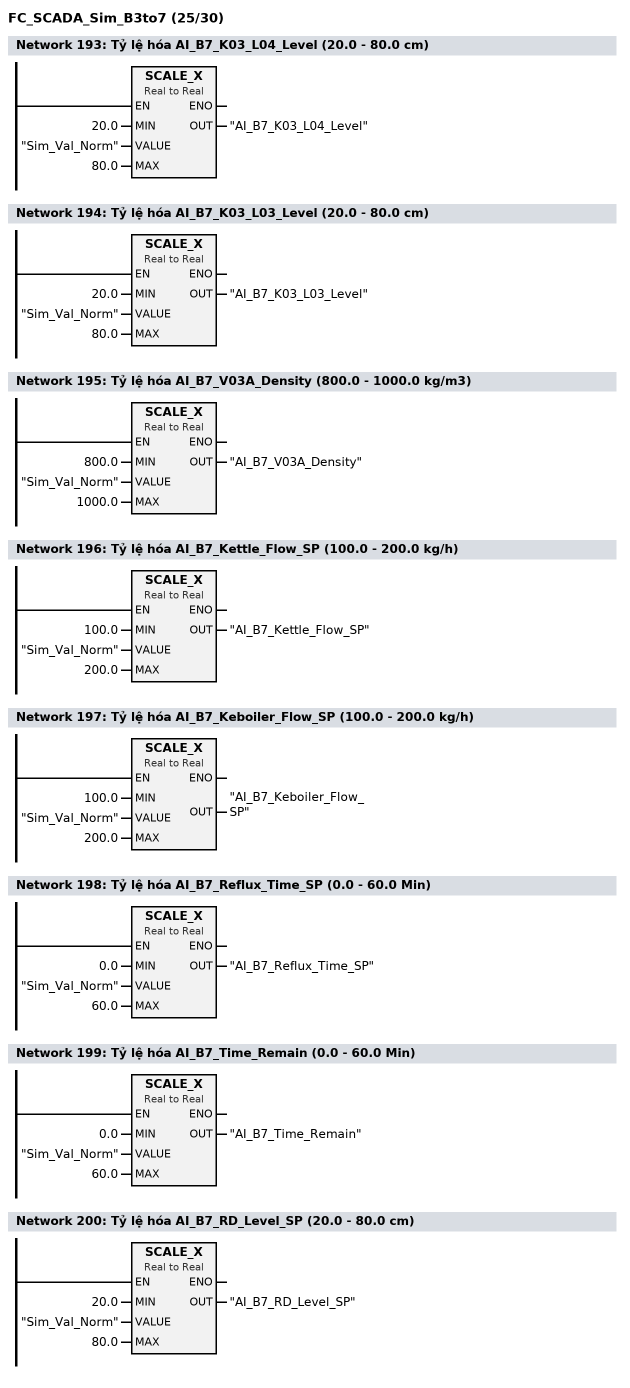
   RUNG wire#powerrail
      { S7_Templates := "[SrcType := Real, DestType := Real]" } Scale(min := 20.0, value := "Sim_Val_Norm", max := 80.0, out => "AI_B7_K03_L04_Level")
   END_RUNG
   // the same network as SCL:
   "AI_B7_K03_L04_Level" := SCALE_X(MIN := 20.0, VALUE := "Sim_Val_Norm", MAX := 80.0);
END_REGION

REGION Network 194: Tỷ lệ hóa AI_B7_K03_L03_Level (20.0 - 80.0 cm)
   RUNG wire#powerrail
      { S7_Templates := "[SrcType := Real, DestType := Real]" } Scale(min := 20.0, value := "Sim_Val_Norm", max := 80.0, out => "AI_B7_K03_L03_Level")
   END_RUNG
   // the same network as SCL:
   "AI_B7_K03_L03_Level" := SCALE_X(MIN := 20.0, VALUE := "Sim_Val_Norm", MAX := 80.0);
END_REGION

REGION Network 195: Tỷ lệ hóa AI_B7_V03A_Density (800.0 - 1000.0 kg/m3)
   RUNG wire#powerrail
      { S7_Templates := "[SrcType := Real, DestType := Real]" } Scale(min := 800.0, value := "Sim_Val_Norm", max := 1000.0, out => "AI_B7_V03A_Density")
   END_RUNG
   // the same network as SCL:
   "AI_B7_V03A_Density" := SCALE_X(MIN := 800.0, VALUE := "Sim_Val_Norm", MAX := 1000.0);
END_REGION

REGION Network 196: Tỷ lệ hóa AI_B7_Kettle_Flow_SP (100.0 - 200.0 kg/h)
   RUNG wire#powerrail
      { S7_Templates := "[SrcType := Real, DestType := Real]" } Scale(min := 100.0, value := "Sim_Val_Norm", max := 200.0, out => "AI_B7_Kettle_Flow_SP")
   END_RUNG
   // the same network as SCL:
   "AI_B7_Kettle_Flow_SP" := SCALE_X(MIN := 100.0, VALUE := "Sim_Val_Norm", MAX := 200.0);
END_REGION

REGION Network 197: Tỷ lệ hóa AI_B7_Keboiler_Flow_SP (100.0 - 200.0 kg/h)
   RUNG wire#powerrail
      { S7_Templates := "[SrcType := Real, DestType := Real]" } Scale(min := 100.0, value := "Sim_Val_Norm", max := 200.0, out => "AI_B7_Keboiler_Flow_SP")
   END_RUNG
   // the same network as SCL:
   "AI_B7_Keboiler_Flow_SP" := SCALE_X(MIN := 100.0, VALUE := "Sim_Val_Norm", MAX := 200.0);
END_REGION

REGION Network 198: Tỷ lệ hóa AI_B7_Reflux_Time_SP (0.0 - 60.0 Min)
   RUNG wire#powerrail
      { S7_Templates := "[SrcType := Real, DestType := Real]" } Scale(min := 0.0, value := "Sim_Val_Norm", max := 60.0, out => "AI_B7_Reflux_Time_SP")
   END_RUNG
   // the same network as SCL:
   "AI_B7_Reflux_Time_SP" := SCALE_X(MIN := 0.0, VALUE := "Sim_Val_Norm", MAX := 60.0);
END_REGION

REGION Network 199: Tỷ lệ hóa AI_B7_Time_Remain (0.0 - 60.0 Min)
   RUNG wire#powerrail
      { S7_Templates := "[SrcType := Real, DestType := Real]" } Scale(min := 0.0, value := "Sim_Val_Norm", max := 60.0, out => "AI_B7_Time_Remain")
   END_RUNG
   // the same network as SCL:
   "AI_B7_Time_Remain" := SCALE_X(MIN := 0.0, VALUE := "Sim_Val_Norm", MAX := 60.0);
END_REGION

REGION Network 200: Tỷ lệ hóa AI_B7_RD_Level_SP (20.0 - 80.0 cm)
   RUNG wire#powerrail
      { S7_Templates := "[SrcType := Real, DestType := Real]" } Scale(min := 20.0, value := "Sim_Val_Norm", max := 80.0, out => "AI_B7_RD_Level_SP")
   END_RUNG
   // the same network as SCL:
   "AI_B7_RD_Level_SP" := SCALE_X(MIN := 20.0, VALUE := "Sim_Val_Norm", MAX := 80.0);
END_REGION

REGION Network 201: Tỷ lệ hóa AI_B7_Reflux_Flow_SP (100.0 - 200.0 L/h)
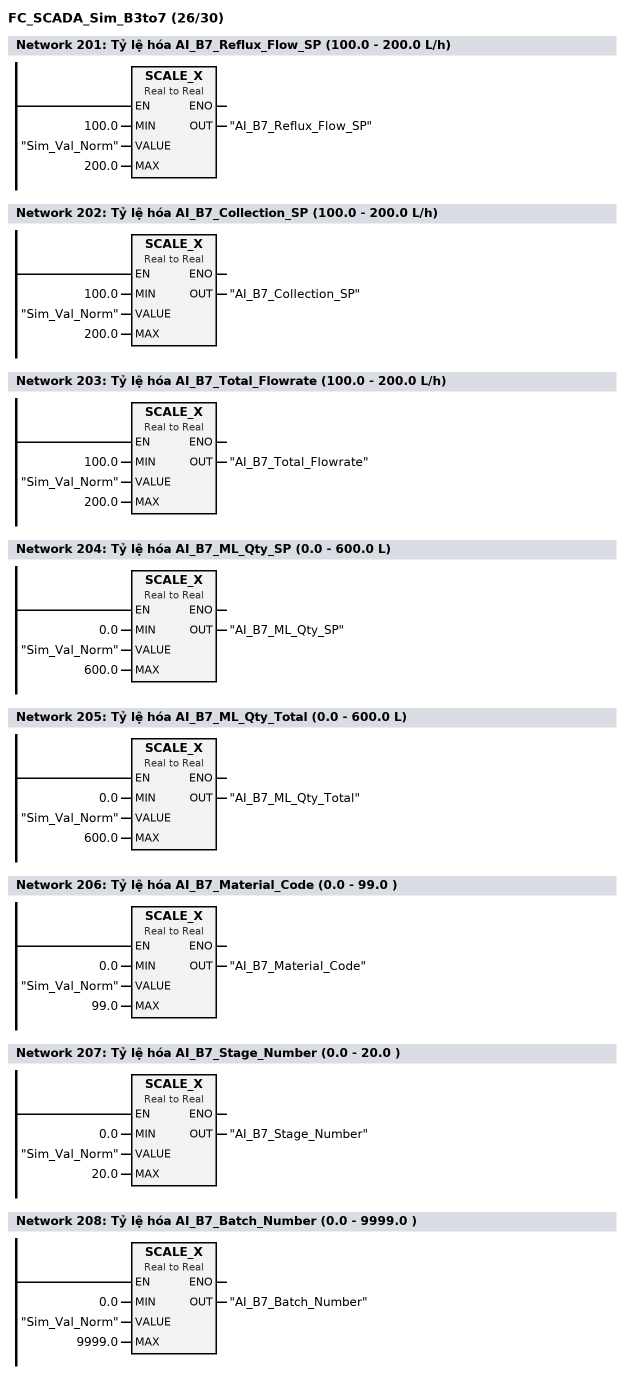
   RUNG wire#powerrail
      { S7_Templates := "[SrcType := Real, DestType := Real]" } Scale(min := 100.0, value := "Sim_Val_Norm", max := 200.0, out => "AI_B7_Reflux_Flow_SP")
   END_RUNG
   // the same network as SCL:
   "AI_B7_Reflux_Flow_SP" := SCALE_X(MIN := 100.0, VALUE := "Sim_Val_Norm", MAX := 200.0);
END_REGION

REGION Network 202: Tỷ lệ hóa AI_B7_Collection_SP (100.0 - 200.0 L/h)
   RUNG wire#powerrail
      { S7_Templates := "[SrcType := Real, DestType := Real]" } Scale(min := 100.0, value := "Sim_Val_Norm", max := 200.0, out => "AI_B7_Collection_SP")
   END_RUNG
   // the same network as SCL:
   "AI_B7_Collection_SP" := SCALE_X(MIN := 100.0, VALUE := "Sim_Val_Norm", MAX := 200.0);
END_REGION

REGION Network 203: Tỷ lệ hóa AI_B7_Total_Flowrate (100.0 - 200.0 L/h)
   RUNG wire#powerrail
      { S7_Templates := "[SrcType := Real, DestType := Real]" } Scale(min := 100.0, value := "Sim_Val_Norm", max := 200.0, out => "AI_B7_Total_Flowrate")
   END_RUNG
   // the same network as SCL:
   "AI_B7_Total_Flowrate" := SCALE_X(MIN := 100.0, VALUE := "Sim_Val_Norm", MAX := 200.0);
END_REGION

REGION Network 204: Tỷ lệ hóa AI_B7_ML_Qty_SP (0.0 - 600.0 L)
   RUNG wire#powerrail
      { S7_Templates := "[SrcType := Real, DestType := Real]" } Scale(min := 0.0, value := "Sim_Val_Norm", max := 600.0, out => "AI_B7_ML_Qty_SP")
   END_RUNG
   // the same network as SCL:
   "AI_B7_ML_Qty_SP" := SCALE_X(MIN := 0.0, VALUE := "Sim_Val_Norm", MAX := 600.0);
END_REGION

REGION Network 205: Tỷ lệ hóa AI_B7_ML_Qty_Total (0.0 - 600.0 L)
   RUNG wire#powerrail
      { S7_Templates := "[SrcType := Real, DestType := Real]" } Scale(min := 0.0, value := "Sim_Val_Norm", max := 600.0, out => "AI_B7_ML_Qty_Total")
   END_RUNG
   // the same network as SCL:
   "AI_B7_ML_Qty_Total" := SCALE_X(MIN := 0.0, VALUE := "Sim_Val_Norm", MAX := 600.0);
END_REGION

REGION Network 206: Tỷ lệ hóa AI_B7_Material_Code (0.0 - 99.0 )
   RUNG wire#powerrail
      { S7_Templates := "[SrcType := Real, DestType := Real]" } Scale(min := 0.0, value := "Sim_Val_Norm", max := 99.0, out => "AI_B7_Material_Code")
   END_RUNG
   // the same network as SCL:
   "AI_B7_Material_Code" := SCALE_X(MIN := 0.0, VALUE := "Sim_Val_Norm", MAX := 99.0);
END_REGION

REGION Network 207: Tỷ lệ hóa AI_B7_Stage_Number (0.0 - 20.0 )
   RUNG wire#powerrail
      { S7_Templates := "[SrcType := Real, DestType := Real]" } Scale(min := 0.0, value := "Sim_Val_Norm", max := 20.0, out => "AI_B7_Stage_Number")
   END_RUNG
   // the same network as SCL:
   "AI_B7_Stage_Number" := SCALE_X(MIN := 0.0, VALUE := "Sim_Val_Norm", MAX := 20.0);
END_REGION

REGION Network 208: Tỷ lệ hóa AI_B7_Batch_Number (0.0 - 9999.0 )
   RUNG wire#powerrail
      { S7_Templates := "[SrcType := Real, DestType := Real]" } Scale(min := 0.0, value := "Sim_Val_Norm", max := 9999.0, out => "AI_B7_Batch_Number")
   END_RUNG
   // the same network as SCL:
   "AI_B7_Batch_Number" := SCALE_X(MIN := 0.0, VALUE := "Sim_Val_Norm", MAX := 9999.0);
END_REGION

REGION Network 209: Tỷ lệ hóa AI_B7_Current_User_ID (0.0 - 999.0 )
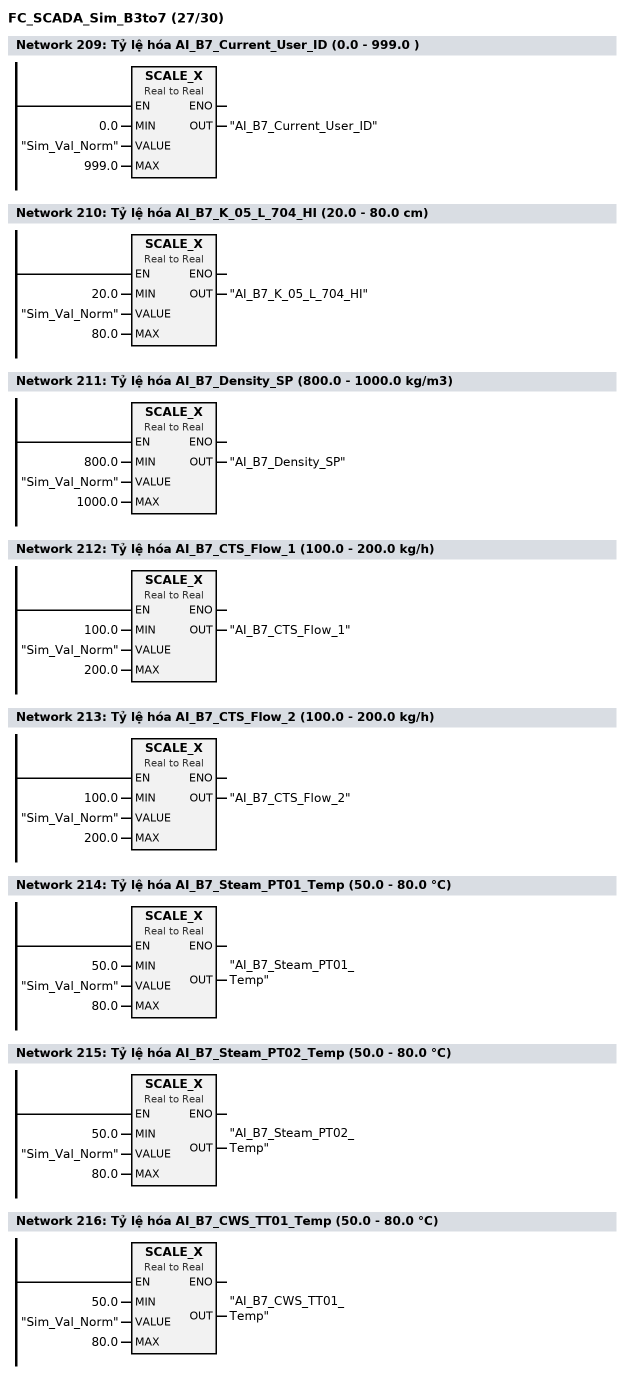
   RUNG wire#powerrail
      { S7_Templates := "[SrcType := Real, DestType := Real]" } Scale(min := 0.0, value := "Sim_Val_Norm", max := 999.0, out => "AI_B7_Current_User_ID")
   END_RUNG
   // the same network as SCL:
   "AI_B7_Current_User_ID" := SCALE_X(MIN := 0.0, VALUE := "Sim_Val_Norm", MAX := 999.0);
END_REGION

REGION Network 210: Tỷ lệ hóa AI_B7_K_05_L_704_HI (20.0 - 80.0 cm)
   RUNG wire#powerrail
      { S7_Templates := "[SrcType := Real, DestType := Real]" } Scale(min := 20.0, value := "Sim_Val_Norm", max := 80.0, out => "AI_B7_K_05_L_704_HI")
   END_RUNG
   // the same network as SCL:
   "AI_B7_K_05_L_704_HI" := SCALE_X(MIN := 20.0, VALUE := "Sim_Val_Norm", MAX := 80.0);
END_REGION

REGION Network 211: Tỷ lệ hóa AI_B7_Density_SP (800.0 - 1000.0 kg/m3)
   RUNG wire#powerrail
      { S7_Templates := "[SrcType := Real, DestType := Real]" } Scale(min := 800.0, value := "Sim_Val_Norm", max := 1000.0, out => "AI_B7_Density_SP")
   END_RUNG
   // the same network as SCL:
   "AI_B7_Density_SP" := SCALE_X(MIN := 800.0, VALUE := "Sim_Val_Norm", MAX := 1000.0);
END_REGION

REGION Network 212: Tỷ lệ hóa AI_B7_CTS_Flow_1 (100.0 - 200.0 kg/h)
   RUNG wire#powerrail
      { S7_Templates := "[SrcType := Real, DestType := Real]" } Scale(min := 100.0, value := "Sim_Val_Norm", max := 200.0, out => "AI_B7_CTS_Flow_1")
   END_RUNG
   // the same network as SCL:
   "AI_B7_CTS_Flow_1" := SCALE_X(MIN := 100.0, VALUE := "Sim_Val_Norm", MAX := 200.0);
END_REGION

REGION Network 213: Tỷ lệ hóa AI_B7_CTS_Flow_2 (100.0 - 200.0 kg/h)
   RUNG wire#powerrail
      { S7_Templates := "[SrcType := Real, DestType := Real]" } Scale(min := 100.0, value := "Sim_Val_Norm", max := 200.0, out => "AI_B7_CTS_Flow_2")
   END_RUNG
   // the same network as SCL:
   "AI_B7_CTS_Flow_2" := SCALE_X(MIN := 100.0, VALUE := "Sim_Val_Norm", MAX := 200.0);
END_REGION

REGION Network 214: Tỷ lệ hóa AI_B7_Steam_PT01_Temp (50.0 - 80.0 °C)
   RUNG wire#powerrail
      { S7_Templates := "[SrcType := Real, DestType := Real]" } Scale(min := 50.0, value := "Sim_Val_Norm", max := 80.0, out => "AI_B7_Steam_PT01_Temp")
   END_RUNG
   // the same network as SCL:
   "AI_B7_Steam_PT01_Temp" := SCALE_X(MIN := 50.0, VALUE := "Sim_Val_Norm", MAX := 80.0);
END_REGION

REGION Network 215: Tỷ lệ hóa AI_B7_Steam_PT02_Temp (50.0 - 80.0 °C)
   RUNG wire#powerrail
      { S7_Templates := "[SrcType := Real, DestType := Real]" } Scale(min := 50.0, value := "Sim_Val_Norm", max := 80.0, out => "AI_B7_Steam_PT02_Temp")
   END_RUNG
   // the same network as SCL:
   "AI_B7_Steam_PT02_Temp" := SCALE_X(MIN := 50.0, VALUE := "Sim_Val_Norm", MAX := 80.0);
END_REGION

REGION Network 216: Tỷ lệ hóa AI_B7_CWS_TT01_Temp (50.0 - 80.0 °C)
   RUNG wire#powerrail
      { S7_Templates := "[SrcType := Real, DestType := Real]" } Scale(min := 50.0, value := "Sim_Val_Norm", max := 80.0, out => "AI_B7_CWS_TT01_Temp")
   END_RUNG
   // the same network as SCL:
   "AI_B7_CWS_TT01_Temp" := SCALE_X(MIN := 50.0, VALUE := "Sim_Val_Norm", MAX := 80.0);
END_REGION

REGION Network 217: Tỷ lệ hóa AI_B7_CWS_TT02_Temp (50.0 - 80.0 °C)
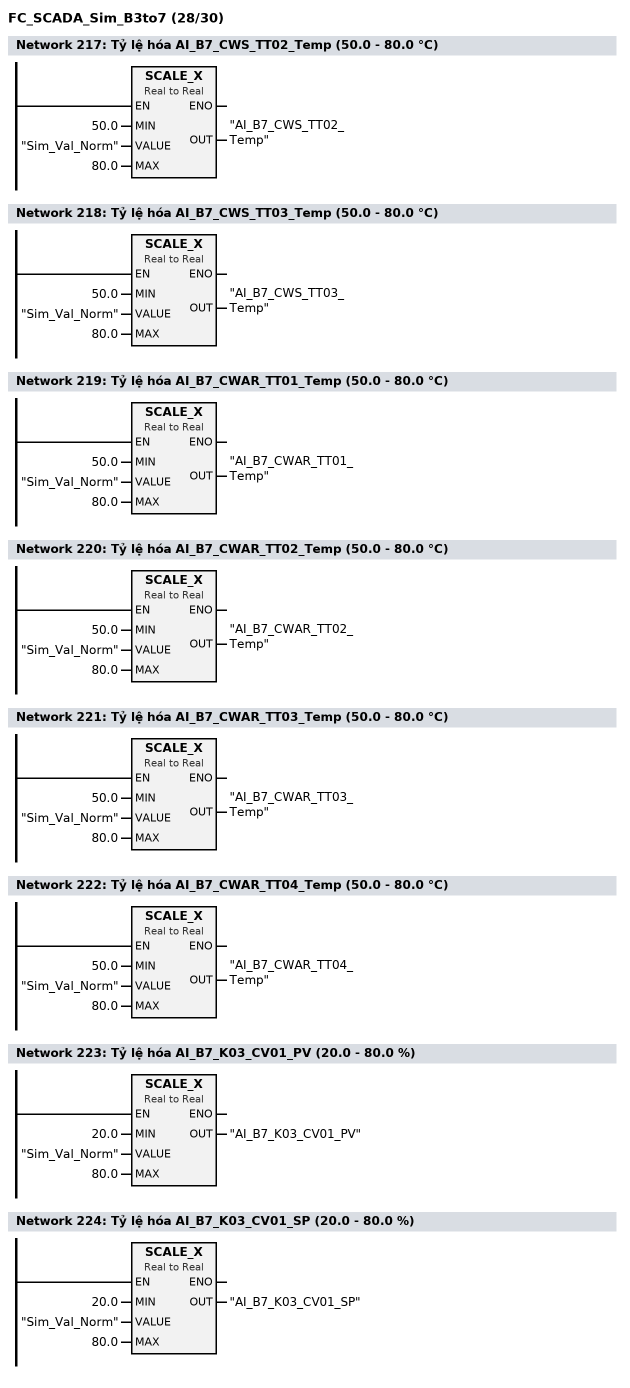
   RUNG wire#powerrail
      { S7_Templates := "[SrcType := Real, DestType := Real]" } Scale(min := 50.0, value := "Sim_Val_Norm", max := 80.0, out => "AI_B7_CWS_TT02_Temp")
   END_RUNG
   // the same network as SCL:
   "AI_B7_CWS_TT02_Temp" := SCALE_X(MIN := 50.0, VALUE := "Sim_Val_Norm", MAX := 80.0);
END_REGION

REGION Network 218: Tỷ lệ hóa AI_B7_CWS_TT03_Temp (50.0 - 80.0 °C)
   RUNG wire#powerrail
      { S7_Templates := "[SrcType := Real, DestType := Real]" } Scale(min := 50.0, value := "Sim_Val_Norm", max := 80.0, out => "AI_B7_CWS_TT03_Temp")
   END_RUNG
   // the same network as SCL:
   "AI_B7_CWS_TT03_Temp" := SCALE_X(MIN := 50.0, VALUE := "Sim_Val_Norm", MAX := 80.0);
END_REGION

REGION Network 219: Tỷ lệ hóa AI_B7_CWAR_TT01_Temp (50.0 - 80.0 °C)
   RUNG wire#powerrail
      { S7_Templates := "[SrcType := Real, DestType := Real]" } Scale(min := 50.0, value := "Sim_Val_Norm", max := 80.0, out => "AI_B7_CWAR_TT01_Temp")
   END_RUNG
   // the same network as SCL:
   "AI_B7_CWAR_TT01_Temp" := SCALE_X(MIN := 50.0, VALUE := "Sim_Val_Norm", MAX := 80.0);
END_REGION

REGION Network 220: Tỷ lệ hóa AI_B7_CWAR_TT02_Temp (50.0 - 80.0 °C)
   RUNG wire#powerrail
      { S7_Templates := "[SrcType := Real, DestType := Real]" } Scale(min := 50.0, value := "Sim_Val_Norm", max := 80.0, out => "AI_B7_CWAR_TT02_Temp")
   END_RUNG
   // the same network as SCL:
   "AI_B7_CWAR_TT02_Temp" := SCALE_X(MIN := 50.0, VALUE := "Sim_Val_Norm", MAX := 80.0);
END_REGION

REGION Network 221: Tỷ lệ hóa AI_B7_CWAR_TT03_Temp (50.0 - 80.0 °C)
   RUNG wire#powerrail
      { S7_Templates := "[SrcType := Real, DestType := Real]" } Scale(min := 50.0, value := "Sim_Val_Norm", max := 80.0, out => "AI_B7_CWAR_TT03_Temp")
   END_RUNG
   // the same network as SCL:
   "AI_B7_CWAR_TT03_Temp" := SCALE_X(MIN := 50.0, VALUE := "Sim_Val_Norm", MAX := 80.0);
END_REGION

REGION Network 222: Tỷ lệ hóa AI_B7_CWAR_TT04_Temp (50.0 - 80.0 °C)
   RUNG wire#powerrail
      { S7_Templates := "[SrcType := Real, DestType := Real]" } Scale(min := 50.0, value := "Sim_Val_Norm", max := 80.0, out => "AI_B7_CWAR_TT04_Temp")
   END_RUNG
   // the same network as SCL:
   "AI_B7_CWAR_TT04_Temp" := SCALE_X(MIN := 50.0, VALUE := "Sim_Val_Norm", MAX := 80.0);
END_REGION

REGION Network 223: Tỷ lệ hóa AI_B7_K03_CV01_PV (20.0 - 80.0 %)
   RUNG wire#powerrail
      { S7_Templates := "[SrcType := Real, DestType := Real]" } Scale(min := 20.0, value := "Sim_Val_Norm", max := 80.0, out => "AI_B7_K03_CV01_PV")
   END_RUNG
   // the same network as SCL:
   "AI_B7_K03_CV01_PV" := SCALE_X(MIN := 20.0, VALUE := "Sim_Val_Norm", MAX := 80.0);
END_REGION

REGION Network 224: Tỷ lệ hóa AI_B7_K03_CV01_SP (20.0 - 80.0 %)
   RUNG wire#powerrail
      { S7_Templates := "[SrcType := Real, DestType := Real]" } Scale(min := 20.0, value := "Sim_Val_Norm", max := 80.0, out => "AI_B7_K03_CV01_SP")
   END_RUNG
   // the same network as SCL:
   "AI_B7_K03_CV01_SP" := SCALE_X(MIN := 20.0, VALUE := "Sim_Val_Norm", MAX := 80.0);
END_REGION

REGION Network 225: Tỷ lệ hóa AI_B7_K03_CV01_CV (20.0 - 80.0 %)
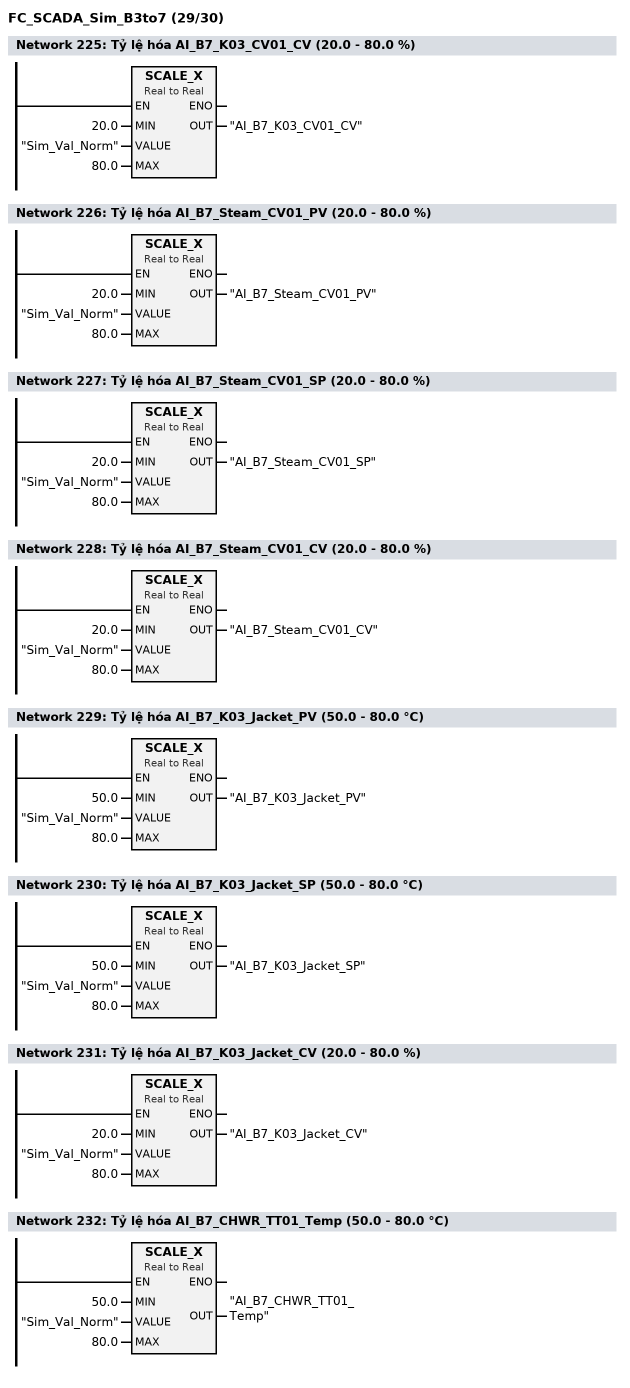
   RUNG wire#powerrail
      { S7_Templates := "[SrcType := Real, DestType := Real]" } Scale(min := 20.0, value := "Sim_Val_Norm", max := 80.0, out => "AI_B7_K03_CV01_CV")
   END_RUNG
   // the same network as SCL:
   "AI_B7_K03_CV01_CV" := SCALE_X(MIN := 20.0, VALUE := "Sim_Val_Norm", MAX := 80.0);
END_REGION

REGION Network 226: Tỷ lệ hóa AI_B7_Steam_CV01_PV (20.0 - 80.0 %)
   RUNG wire#powerrail
      { S7_Templates := "[SrcType := Real, DestType := Real]" } Scale(min := 20.0, value := "Sim_Val_Norm", max := 80.0, out => "AI_B7_Steam_CV01_PV")
   END_RUNG
   // the same network as SCL:
   "AI_B7_Steam_CV01_PV" := SCALE_X(MIN := 20.0, VALUE := "Sim_Val_Norm", MAX := 80.0);
END_REGION

REGION Network 227: Tỷ lệ hóa AI_B7_Steam_CV01_SP (20.0 - 80.0 %)
   RUNG wire#powerrail
      { S7_Templates := "[SrcType := Real, DestType := Real]" } Scale(min := 20.0, value := "Sim_Val_Norm", max := 80.0, out => "AI_B7_Steam_CV01_SP")
   END_RUNG
   // the same network as SCL:
   "AI_B7_Steam_CV01_SP" := SCALE_X(MIN := 20.0, VALUE := "Sim_Val_Norm", MAX := 80.0);
END_REGION

REGION Network 228: Tỷ lệ hóa AI_B7_Steam_CV01_CV (20.0 - 80.0 %)
   RUNG wire#powerrail
      { S7_Templates := "[SrcType := Real, DestType := Real]" } Scale(min := 20.0, value := "Sim_Val_Norm", max := 80.0, out => "AI_B7_Steam_CV01_CV")
   END_RUNG
   // the same network as SCL:
   "AI_B7_Steam_CV01_CV" := SCALE_X(MIN := 20.0, VALUE := "Sim_Val_Norm", MAX := 80.0);
END_REGION

REGION Network 229: Tỷ lệ hóa AI_B7_K03_Jacket_PV (50.0 - 80.0 °C)
   RUNG wire#powerrail
      { S7_Templates := "[SrcType := Real, DestType := Real]" } Scale(min := 50.0, value := "Sim_Val_Norm", max := 80.0, out => "AI_B7_K03_Jacket_PV")
   END_RUNG
   // the same network as SCL:
   "AI_B7_K03_Jacket_PV" := SCALE_X(MIN := 50.0, VALUE := "Sim_Val_Norm", MAX := 80.0);
END_REGION

REGION Network 230: Tỷ lệ hóa AI_B7_K03_Jacket_SP (50.0 - 80.0 °C)
   RUNG wire#powerrail
      { S7_Templates := "[SrcType := Real, DestType := Real]" } Scale(min := 50.0, value := "Sim_Val_Norm", max := 80.0, out => "AI_B7_K03_Jacket_SP")
   END_RUNG
   // the same network as SCL:
   "AI_B7_K03_Jacket_SP" := SCALE_X(MIN := 50.0, VALUE := "Sim_Val_Norm", MAX := 80.0);
END_REGION

REGION Network 231: Tỷ lệ hóa AI_B7_K03_Jacket_CV (20.0 - 80.0 %)
   RUNG wire#powerrail
      { S7_Templates := "[SrcType := Real, DestType := Real]" } Scale(min := 20.0, value := "Sim_Val_Norm", max := 80.0, out => "AI_B7_K03_Jacket_CV")
   END_RUNG
   // the same network as SCL:
   "AI_B7_K03_Jacket_CV" := SCALE_X(MIN := 20.0, VALUE := "Sim_Val_Norm", MAX := 80.0);
END_REGION

REGION Network 232: Tỷ lệ hóa AI_B7_CHWR_TT01_Temp (50.0 - 80.0 °C)
   RUNG wire#powerrail
      { S7_Templates := "[SrcType := Real, DestType := Real]" } Scale(min := 50.0, value := "Sim_Val_Norm", max := 80.0, out => "AI_B7_CHWR_TT01_Temp")
   END_RUNG
   // the same network as SCL:
   "AI_B7_CHWR_TT01_Temp" := SCALE_X(MIN := 50.0, VALUE := "Sim_Val_Norm", MAX := 80.0);
END_REGION

REGION Network 233: Tỷ lệ hóa AI_B7_CHWR_TT02_Temp (50.0 - 80.0 °C)
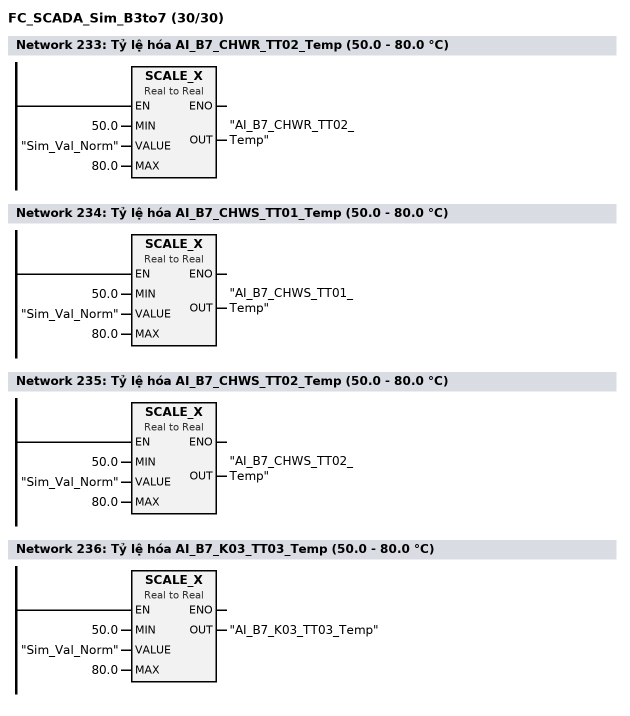
   RUNG wire#powerrail
      { S7_Templates := "[SrcType := Real, DestType := Real]" } Scale(min := 50.0, value := "Sim_Val_Norm", max := 80.0, out => "AI_B7_CHWR_TT02_Temp")
   END_RUNG
   // the same network as SCL:
   "AI_B7_CHWR_TT02_Temp" := SCALE_X(MIN := 50.0, VALUE := "Sim_Val_Norm", MAX := 80.0);
END_REGION

REGION Network 234: Tỷ lệ hóa AI_B7_CHWS_TT01_Temp (50.0 - 80.0 °C)
   RUNG wire#powerrail
      { S7_Templates := "[SrcType := Real, DestType := Real]" } Scale(min := 50.0, value := "Sim_Val_Norm", max := 80.0, out => "AI_B7_CHWS_TT01_Temp")
   END_RUNG
   // the same network as SCL:
   "AI_B7_CHWS_TT01_Temp" := SCALE_X(MIN := 50.0, VALUE := "Sim_Val_Norm", MAX := 80.0);
END_REGION

REGION Network 235: Tỷ lệ hóa AI_B7_CHWS_TT02_Temp (50.0 - 80.0 °C)
   RUNG wire#powerrail
      { S7_Templates := "[SrcType := Real, DestType := Real]" } Scale(min := 50.0, value := "Sim_Val_Norm", max := 80.0, out => "AI_B7_CHWS_TT02_Temp")
   END_RUNG
   // the same network as SCL:
   "AI_B7_CHWS_TT02_Temp" := SCALE_X(MIN := 50.0, VALUE := "Sim_Val_Norm", MAX := 80.0);
END_REGION

REGION Network 236: Tỷ lệ hóa AI_B7_K03_TT03_Temp (50.0 - 80.0 °C)
   RUNG wire#powerrail
      { S7_Templates := "[SrcType := Real, DestType := Real]" } Scale(min := 50.0, value := "Sim_Val_Norm", max := 80.0, out => "AI_B7_K03_TT03_Temp")
   END_RUNG
   // the same network as SCL:
   "AI_B7_K03_TT03_Temp" := SCALE_X(MIN := 50.0, VALUE := "Sim_Val_Norm", MAX := 80.0);
END_REGION
END_FUNCTION
